(* CODESYS project SPT_NC_Homing.library
   Company: Beckhoff Automation LLC
   DefaultNamespace: SPT_NCHoming
   Version: 3.0.0
   Placeholder: SPT NC Homing
   Title: SPT NC Homing

Project tree, tasks and I/O mapping:
  libraries: SPT Base Types, * (Beckhoff Automation LLC); SPT NC Axis, * (Beckhoff Automation LLC); Tc2_MC2, * (Beckhoff Automation GmbH); Tc3_MC2_AdvancedHoming, * (Beckhoff Automation GmbH); Tc3_Module, * (Beckhoff Automation GmbH); Tc3_System, * (Beckhoff Automation GmbH)
  DUTs/
    data type ST_StepBlockLagBasedParameters
  Function Blocks/
    function block FB_HomeRoutine_HardStop [ST]: Axis, Execute, HomePosition, Parameters
    function block FB_HomeRoutine_SetPosition [ST]: Axis, Execute, HomePosition
    function block FB_HomeRoutine_SetZeroHere [ST]: Axis, Execute
  Project Information/
    function F_GetCompany [ST]
    function F_GetTitle [ST]
    function F_GetVersion [ST]
  Version/
    global variables Global_Version
*)

// DUTs/ST_StepBlockLagBasedParameters
TYPE ST_StepBlockLagBasedParameters :
    STRUCT
        Direction              : MC_Home_Direction := mcNegativeDirection;
        Velocity               : LREAL             := 10;
        Acceleration           : LREAL             := 100;
        Deceleration           : LREAL             := 100;
        Jerk                   : LREAL             := 1000;
        DetectionVelocityLimit : LREAL             := 5;
        DetectionVelocityTime  : TIME              := T#500MS;
        TimeLimit              : TIME;
        DistanceLimit          : LREAL;
        TorqueLimit            : LREAL            := 10;
        LagLimit               : LREAL            := 10;
        Options                : ST_Home_Options3 := (InstantLagReduction := TRUE);
    END_STRUCT
END_TYPE

// Version/Global_Version
{attribute 'TcGenerated'}
{attribute 'no-analysis'}
{attribute 'linkalways'}
// This function has been automatically generated from the project information.
VAR_GLOBAL CONSTANT
	{attribute 'const_non_replaced'}
	stLibVersion_SPT_NC_Homing : ST_LibVersion := (iMajor := 3, iMinor := 0, iBuild := 0, iRevision := 0, nFlags := 1, sVersion := '3.0.0');
END_VAR

// Function Blocks/FB_HomeRoutine_HardStop
FUNCTION_BLOCK FINAL FB_HomeRoutine_HardStop EXTENDS FB_BaseFB IMPLEMENTS I_MotionSequence
VAR
    _Axis : I_BasicAxis;
END_VAR

VAR
    MCStepBlock    : MC_StepBlockLagBasedDetection;
    MCHomeDirect   : MC_HomeDirect;
	MCReset			: MC_Reset;
    MCAbortHoming  : MC_AbortHoming;
    AxisParameters : MC_HomingParameter;
    _Parameters    : ST_StepBlockLagBasedParameters;
    _HomePosition  : LREAL;
    SequenceStep   : UDINT;
END_VAR

CASE SequenceStep OF
    10:
        MCStepBlock(Axis                   := _Axis.Axis,
                    Parameter              := AxisParameters,
                    Execute                := TRUE,
                    Direction              := _Parameters.Direction,
                    Velocity               := _Parameters.Velocity,
                    Acceleration           := _Parameters.Acceleration,
                    Deceleration           := _Parameters.Deceleration,
                    Jerk                   := _Parameters.Jerk,
                    DetectionVelocityLimit := _Parameters.DetectionVelocityLimit,
                    DetectionVelocityTime  := _Parameters.DetectionVelocityTime,
                    TimeLimit              := _Parameters.TimeLimit,
                    DistanceLimit          := _Parameters.DistanceLimit,
                    TorqueLimit            := _Parameters.TorqueLimit,
                    LagLimit               := _Parameters.LagLimit,
                    Options                := _Parameters.Options);

        IF NOT MCStepBlock.Busy THEN
            IF MCStepBlock.Error THEN
                _Error       := TRUE;
                _ErrorID     := MCStepBlock.ErrorID;
                SequenceStep := 999;
            ELSE
                //No error occurred
                SequenceStep := SequenceStep + 10;
            END_IF

            MCStepBlock(Axis := _Axis.Axis, Parameter := AxisParameters, Execute := FALSE);
        END_IF
    20:
        MCHomeDirect(Axis        := _Axis.Axis,
                     Parameter   := AxisParameters,
                     Execute     := TRUE,
                     SetPosition := _HomePosition);

        IF NOT MCHomeDirect.Busy THEN
            IF MCHomeDirect.Error THEN
                _Error       := TRUE;
                _ErrorID     := MCHomeDirect.ErrorID;
                SequenceStep := 999;
            END_IF

            //Done
            SequenceStep := 0;
            MCHomeDirect(Axis := _Axis.Axis, Parameter := AxisParameters, Execute := FALSE);
        END_IF
    999:
        //An error occurred above--clear out position lag so we don't fault the axis with AbortHoming
        MCReset(Axis := _Axis.Axis, Execute := TRUE);
        IF NOT MCReset.Busy THEN
            //If this errors there's not much we can do about it
            SequenceStep := 1000;
            MCReset(Axis := _Axis.Axis, Execute := FALSE);
        END_IF
    1000:
        MCAbortHoming(Axis := _Axis.Axis, Parameter := AxisParameters, Execute := TRUE);
        IF NOT MCAbortHoming.Busy THEN
            IF MCAbortHoming.Error THEN
                _Error       := TRUE;
                _ErrorID     := MCAbortHoming.ErrorID;
                SequenceStep := 0;
            ELSE
                //No error occurred
                SequenceStep := 0;
            END_IF

            MCAbortHoming(Axis := _Axis.Axis, Parameter := AxisParameters, Execute := FALSE);
        END_IF
END_CASE

_Busy := SequenceStep <> 0;

PROPERTY Axis : I_BasicAxis
GET
Axis := _Axis;
END_GET
SET
_Axis := Axis;
END_SET
END_PROPERTY

METHOD PUBLIC Execute : BOOL
IF (_Axis = 0) OR _Busy THEN
    RETURN;
END_IF

_Busy        := TRUE;
_Error       := FALSE;
_ErrorID     := 0;
SequenceStep := 10;
Execute      := TRUE;
END_METHOD

PROPERTY HomePosition : LREAL
GET
HomePosition := _HomePosition;
END_GET
SET
_HomePosition := HomePosition;
END_SET
END_PROPERTY

PROPERTY Parameters : ST_StepBlockLagBasedParameters
GET
Parameters := _Parameters;
END_GET
SET
_Parameters := Parameters;
END_SET
END_PROPERTY

END_FUNCTION_BLOCK

// Function Blocks/FB_HomeRoutine_SetPosition
FUNCTION_BLOCK FINAL FB_HomeRoutine_SetPosition EXTENDS FB_BaseFB IMPLEMENTS I_MotionSequence
VAR_INPUT
END_VAR
VAR_OUTPUT
END_VAR
VAR
    _Axis : I_BasicAxis;
END_VAR

VAR
    MCSetPosition : MC_SetPosition;
END_VAR

MCSetPosition(Axis := _Axis.Axis, Busy => _Busy);

IF NOT MCSetPosition.Busy THEN
    IF MCSetPosition.Error THEN
        _Error   := TRUE;
        _ErrorID := MCSetPosition.ErrorID;
    END_IF

    MCSetPosition(Axis := _Axis.Axis, Execute := FALSE);
END_IF

PROPERTY Axis : I_BasicAxis
GET
Axis := _Axis;
END_GET
SET
_Axis := Axis;
END_SET
END_PROPERTY

METHOD PUBLIC Execute : BOOL
IF (_Axis = 0) THEN
    RETURN;
END_IF

MCSetPosition(Axis := _Axis.Axis, Execute := TRUE, Mode := FALSE);

_Error   := FALSE;
_ErrorID := 0;

Execute := TRUE;
END_METHOD

PROPERTY HomePosition : LREAL
GET
HomePosition := MCSetPosition.Position;
END_GET
SET
MCSetPosition.Position := HomePosition;
END_SET
END_PROPERTY

END_FUNCTION_BLOCK

// Function Blocks/FB_HomeRoutine_SetZeroHere
FUNCTION_BLOCK FINAL FB_HomeRoutine_SetZeroHere EXTENDS FB_BaseFB IMPLEMENTS I_MotionSequence
VAR_INPUT
END_VAR
VAR_OUTPUT
END_VAR
VAR
    _Axis : I_BasicAxis;
END_VAR

VAR
    MCSetPosition : MC_SetPosition;
END_VAR

MCSetPosition(Axis := _Axis.Axis, Busy => _Busy);

IF NOT MCSetPosition.Busy THEN
    IF MCSetPosition.Error THEN
        _Error   := TRUE;
        _ErrorID := MCSetPosition.ErrorID;
    END_IF

    MCSetPosition(Axis := _Axis.Axis, Execute := FALSE);
END_IF

PROPERTY Axis : I_BasicAxis
GET
Axis := _Axis;
END_GET
SET
_Axis := Axis;
END_SET
END_PROPERTY

METHOD PUBLIC Execute : BOOL
IF (_Axis = 0) THEN
    RETURN;
END_IF

MCSetPosition(Axis := _Axis.Axis, Execute := TRUE, Position := 0.0, Mode := FALSE);

_Error   := FALSE;
_ErrorID := 0;

Execute := TRUE;
END_METHOD

END_FUNCTION_BLOCK

// Project Information/F_GetCompany
// This function has been automatically generated from the project information.
{attribute 'signature_flag' := '1073741824'}
{attribute 'TcGenerated'}
{attribute 'no-analysis'}
FUNCTION F_GetCompany : WSTRING
VAR_INPUT
	
END_VAR

F_GetCompany := "Beckhoff Automation LLC";

END_FUNCTION

// Project Information/F_GetTitle
// This function has been automatically generated from the project information.
{attribute 'signature_flag' := '1073741824'}
{attribute 'TcGenerated'}
{attribute 'no-analysis'}
FUNCTION F_GetTitle : WSTRING
VAR_INPUT
	
END_VAR

F_GetTitle := "SPT NC Homing";

END_FUNCTION

// Project Information/F_GetVersion
// This function has been automatically generated from the project information.
{attribute 'signature_flag' := '1073741824'}
{attribute 'TcGenerated'}
{attribute 'no-analysis'}
FUNCTION F_GetVersion : ST_LibVersion
VAR_INPUT
	
END_VAR

F_GetVersion.iMajor := 3;
F_GetVersion.iMinor := 0;
F_GetVersion.iBuild := 0;
F_GetVersion.iRevision := 0;
F_GetVersion.sVersion := '3.0.0';
F_GetVersion.nFlags := 1;

END_FUNCTION
